PROGRAM PRG_HmiStatus
VAR
    fbBlinkTimer    : TON;
    bBlinkTimerQOld : BOOL;
    bFlash          : BOOL;
    fbEL6910Diagnostics : FB_EL6910Diagnostics;
    uiHeatStakeReasonNestId : UINT;
    bHeatStakeReasonRejectPending : BOOL;
END_VAR

// Same 500 ms toggle used by the validated Silicone Station banner.
fbBlinkTimer(IN := NOT fbBlinkTimer.Q, PT := T#500MS);

IF fbBlinkTimer.Q AND NOT bBlinkTimerQOld THEN
    GVL_HMI.bBlink_1Hz := NOT GVL_HMI.bBlink_1Hz;
END_IF

bBlinkTimerQOld := fbBlinkTimer.Q;
bFlash := GVL_HMI.bBlink_1Hz;

GVL_HMI.stStatus.eMachineState := GVL_MASTER.stStatus.eMachineState;
GVL_HMI.stStatus.eIndexState := GVL_MASTER.stStatus.eIndexState;
GVL_HMI.stStatus.eIndexPosition := GVL_MASTER.stInputs.eIndexPosition;
GVL_HMI.stStatus.bReady := GVL_MASTER.stStatus.bReady;
GVL_HMI.stStatus.bBusy := GVL_MASTER.stStatus.bBusy;
GVL_HMI.stStatus.bFaulted := GVL_MASTER.stStatus.bFaulted;
GVL_HMI.stStatus.bTwoHandsSafe := GVL_MASTER.stInputs.bTwoHandsSafe;
// Physical operator-nest part-present indication.
// This is intentionally NOT derived from nest tracking/result state.
// It follows the real sensor immediately whenever the operator places/removes
// a part in the nest currently located at the operator position.
GVL_HMI.stStatus.bLoadingStationEaglePresent :=GVL_IO.stInputs.bLoadingStationEaglePresent;
GVL_HMI.stStatus.bLoadingStationPbupPresent := GVL_IO.stInputs.bLoadingStationPbupPresent;
GVL_HMI.stStatus.bRejectChutePartPresent := GVL_MASTER.stInputs.bRejectChutePartPresent;
GVL_HMI.stStatus.bHeatStakeEaglePresent := GVL_MASTER.stInputs.bHeatStakeEaglePresent;
GVL_HMI.stStatus.bHeatStakePatchPresent := GVL_MASTER.stInputs.bHeatStakePatchPresent;
GVL_HMI.stStatus.bPbupMagnetPresent := GVL_MASTER.stInputs.bPbupMagnetPresent;
GVL_HMI.stStatus.bIndexReady := GVL_MASTER.stInputs.bIndexReady;
GVL_HMI.stStatus.bIndexLocked := GVL_MASTER.stInputs.bIndexLocked;
GVL_HMI.stStatus.bIndexCompletedSensor := GVL_MASTER.stInputs.bIndexCompletedSensor;
GVL_HMI.stStatus.bMainDoorClosed := GVL_MASTER.stInputs.bMainDoorClosed;
GVL_HMI.stStatus.bMainDoorLocked := GVL_MASTER.stInputs.bMainDoorLocked;
GVL_HMI.stStatus.bStartButtonActive := GVL_MASTER.stInputs.bStartButton;
GVL_HMI.stStatus.bStopButtonActive := GVL_MASTER.stInputs.bStopButton;
GVL_HMI.stStatus.bResetButtonActive := GVL_MASTER.stInputs.bResetButton;
GVL_HMI.stStatus.bStartButtonLamp := GVL_MASTER.stOutputs.bLedStart;
GVL_HMI.stStatus.bUp24VPowerSupplyOk := GVL_MASTER.stInputs.bUp24VPowerSupplyOk;
GVL_HMI.stStatus.bUs24VPowerSupplyOk := GVL_MASTER.stInputs.bUs24VPowerSupplyOk;
GVL_HMI.stStatus.b48VPowerSupplyOk := GVL_MASTER.stInputs.b48VPowerSupplyOk;
GVL_HMI.stStatus.bMainDoorDiagnosticOk := GVL_MASTER.stInputs.bMainDoorDiagnosticOk;
GVL_HMI.stStatus.bMs6FeedbackOk := GVL_MASTER.stInputs.bMs6FeedbackOk;
GVL_HMI.stStatus.bAirExhausted := GVL_MASTER.stInputs.bAirExhausted;
GVL_HMI.stStatus.bLeftFlapSafe := GVL_MASTER.stInputs.stSafety.bLeftFlapSafe;
GVL_HMI.stStatus.bRightFlapSafe := GVL_MASTER.stInputs.stSafety.bRightFlapSafe;
GVL_HMI.stStatus.bEnableSettings := GVL_MASTER.stStatus.bEnableSetting;
GVL_HMI.stStatus.bAllStationsCommissioned := GVL_MASTER.stStatus.bAllStationsCommissioned;
GVL_HMI.stStatus.bAutoCycleAllowed := GVL_MASTER.stStatus.bAutoCycleAllowed;
GVL_HMI.stStatus.bPatchSupportRetracted := FALSE; // Retired status; no sensor is fitted.
GVL_HMI.stStatus.bPatchSupportExtended := FALSE; // Retired status; no sensor is fitted.


GVL_HMI.stStatus.bNest1Blocked := NOT GVL_Persistent.aNestEnabled[1];
GVL_HMI.stStatus.bNest2Blocked := NOT GVL_Persistent.aNestEnabled[2];
GVL_HMI.stStatus.bNest3Blocked := NOT GVL_Persistent.aNestEnabled[3];
GVL_HMI.stStatus.bNest4Blocked := NOT GVL_Persistent.aNestEnabled[4];

GVL_HMI.stStatus.bDisabledNestPartIndexBlocked := GVL_MASTER.stStatus.bDisabledNestPartIndexBlocked;
GVL_HMI.stStatus.bDisabledNestPartPopupRequest :=GVL_MASTER.stStatus.bDisabledNestPartPopupRequest;
GVL_HMI.stStatus.uiDisabledNestPartPopupNestId :=GVL_MASTER.stStatus.uiDisabledNestPartPopupNestId;

GVL_HMI.stStatus.bRejectChuteFullLatched :=GVL_MASTER.stStatus.bRejectChuteFullLatched;
GVL_HMI.stStatus.bRejectChutePopupRequest :=GVL_MASTER.stStatus.bRejectChutePopupRequest;
GVL_HMI.stStatus.bRejectChuteStopRequest :=GVL_MASTER.stStatus.bRejectChuteStopRequest;
GVL_HMI.stStatus.bRejectChuteResetBlocked :=GVL_MASTER.stStatus.bRejectChuteResetBlocked;

GVL_HMI.stStatus.sRejectChutePopupMessage :=
    'Reject chute is full. Empty the reject chute and press Acknowledge.';

GVL_HMI.stStatus.bHeatStakeHeadUp := GVL_MASTER.stStatus.bHeatStakeHeadUp;
GVL_HMI.stStatus.bHeatStakeHeadDown := GVL_MASTER.stStatus.bHeatStakeHeadDown;
GVL_HMI.stStatus.bHeatStakeHeadDownTimeoutFault := GVL_MASTER.stStatus.bHeatStakeHeadDownTimeoutFault;
GVL_HMI.stStatus.bHeatStakeHeadUpTimeoutFault := GVL_MASTER.stStatus.bHeatStakeHeadUpTimeoutFault;
GVL_HMI.stStatus.bHeatStakeHeadSensorConflictFault := GVL_MASTER.stStatus.bHeatStakeHeadSensorConflictFault;

// Use the same TC3/head criterion as the machine's hot-door lock demand.
GVL_HMI.bUnlockDoorVisible :=
    (GVL_MASTER.stStatus.eMachineState = E_MachineState.Stopped)
    AND GVL_MASTER.stStatus.stMainDoorLock.bLockRequest
    AND NOT (GVL_MASTER.stStatus.stHeatStakeTemperature.rOverTempTemperatureC <
        GVL_Config.rMainDoorHotTemperatureLimitC);
// A stale hot-door popup must not remain open once the head cools or the state changes.
IF NOT GVL_HMI.bUnlockDoorVisible THEN
    GVL_HMI.bUnlockDoorPopupRequest := FALSE;
END_IF


IF (GVL_MASTER.stStatus.uiDisabledNestPartPopupNestId >= 1)
    AND (GVL_MASTER.stStatus.uiDisabledNestPartPopupNestId <= 4)
THEN
    GVL_HMI.stStatus.sDisabledNestPartPopupMessage :=
        CONCAT(
            CONCAT(
                'Nest ',
                UINT_TO_STRING(GVL_MASTER.stStatus.uiDisabledNestPartPopupNestId)
            ),
            ' is disabled. Remove the part from this nest before indexing.'
        );
ELSE
    GVL_HMI.stStatus.sDisabledNestPartPopupMessage :=
        'A disabled nest contains a part. Remove the part before indexing.';
END_IF

GVL_HMI.stStatus.stPatchDispense := GVL_MASTER.stStatus.stPatchDispense;
// Display aggregate Patch faults, including feeding/motion, without changing control state.
GVL_HMI.stStatus.stPatchDispense.bFault :=
    GVL_MASTER.stStatus.stPatchDispense.bFault
    OR GVL_Motion.stPatchFeedStatus.bFault
    OR GVL_Motion.AxisDriveMotor.bError;
IF GVL_MASTER.stStatus.eMachineState = E_MachineState.Manual THEN
    // Continuous UP holding at HOME is idle; actual manual actions are busy.
    GVL_HMI.stStatus.stPatchDispense.bBusy :=
        GVL_MASTER.stStatus.stPatchDispense.bBusy
        OR NOT GVL_MASTER.stStatus.stPatchDispense.bHome
        OR GVL_Motion.stPatchFeedStatus.bBusy
        OR GVL_Motion.AxisDriveMotor.bMoving
        OR GVL_MASTER.stOutputs.bPatchVerticalDown
        OR GVL_MASTER.stOutputs.bPatchDispenserAir;
    GVL_HMI.stStatus.stPatchDispense.bReady :=
        GVL_MASTER.stStatus.stPatchDispense.bCommissioned
        AND GVL_MASTER.stStatus.stPatchDispense.bHome
        AND NOT GVL_HMI.stStatus.stPatchDispense.bBusy
        AND NOT GVL_HMI.stStatus.stPatchDispense.bFault;
END_IF
// ReadyToStart indication accepts the deliberately disabled, idle M1 axis.
// This does not change FB readiness, motion enable or sequence start permissives.
IF GVL_MASTER.stStatus.eMachineState = E_MachineState.ReadyToStart THEN
    GVL_HMI.stStatus.stPatchDispense.bReady :=
        GVL_MASTER.stStatus.stPatchDispense.bCommissioned
        AND (GVL_MASTER.stStatus.stPatchDispense.eState = E_PatchStationState.Ready)
        AND GVL_MASTER.stStatus.stPatchDispense.bHome
        AND NOT GVL_MASTER.stStatus.stPatchDispense.bBusy
        AND NOT GVL_HMI.stStatus.stPatchDispense.bFault
        AND GVL_MASTER.stInputs.stSafety.bSafetyOk
        AND GVL_MASTER.stInputs.stSafety.bMotionSafetyPermitted
        AND GVL_MASTER.stInputs.bMainDoorClosed
        AND GVL_Safety.bAirSupplySafe
        AND NOT GVL_Motion.stPatchFeedStatus.bBusy
        AND NOT GVL_Motion.AxisDriveMotor.bMoving
        AND NOT GVL_Motion.AxisDriveMotor.Axis.Status.ErrorStop
        AND (GVL_Motion.AxisDriveMotor.Axis.NcToPlc.AxisId <> 0)
        AND (GVL_Motion.AxisDriveMotor.bStandstill
            OR GVL_Motion.AxisDriveMotor.Axis.Status.Disabled);
END_IF
GVL_HMI.stStatus.stHeatStake := GVL_MASTER.stStatus.stHeatStake;
GVL_HMI.stStatus.stHeatStakeTemperature := GVL_MASTER.stStatus.stHeatStakeTemperature;
GVL_HMI.stStatus.stHeatStakeProcess := GVL_MASTER.stStatus.stHeatStakeProcess;
GVL_HMI.stStatus.stHeatStakeProcessSettings := GVL_Persistent.stHeatStakeProcessSettings;
GVL_HMI.stStatus.bHeatStakeProcessSettingsWriteBusy := PRG_HeatStakeProcessSettings.bWriteBusy;
GVL_HMI.stStatus.bHeatStakeProcessSettingsWriteError := PRG_HeatStakeProcessSettings.bWriteError;
GVL_HMI.stStatus.udiHeatStakeProcessSettingsWriteErrorId := PRG_HeatStakeProcessSettings.udiWriteErrorId;
GVL_HMI.stStatus.stHeatStakeTemperatureSettings := GVL_Persistent.stHeatStakeTemperatureSettings;
GVL_HMI.stStatus.bHeatStakeSettingsApplyAccepted := PRG_HeatStakeTemperatureSettings.bApplyAccepted;
GVL_HMI.stStatus.bHeatStakeSettingsApplyRejected := PRG_HeatStakeTemperatureSettings.bApplyRejected;
GVL_HMI.stStatus.bHeatStakeSettingsWriteBusy := PRG_HeatStakeTemperatureSettings.bWriteBusy;
GVL_HMI.stStatus.bHeatStakeSettingsWriteError := PRG_HeatStakeTemperatureSettings.bWriteError;
GVL_HMI.stStatus.bHeatStakeSettingsSaveSuccessful := PRG_HeatStakeTemperatureSettings.bSaveSuccessful;
GVL_HMI.stStatus.bHeatStakeSettingsSaveFailed := PRG_HeatStakeTemperatureSettings.bSaveFailed;
GVL_HMI.stStatus.sHeatStakeSettingsApplyRejectReason := PRG_HeatStakeTemperatureSettings.sApplyRejectReason;
GVL_HMI.stStatus.udiHeatStakeSettingsWriteErrorId := PRG_HeatStakeTemperatureSettings.udiWriteErrorId;

// Manual-mode indexer station/nest display.
GVL_HMI.stStatus.uiPatchDispenseNestId := GVL_MASTER.stStatus.uiPatchDispenseNestId;
GVL_HMI.stStatus.uiHeatStakeNestId := GVL_MASTER.stStatus.uiHeatStakeNestId;
GVL_HMI.stStatus.uiVisionNestId := GVL_MASTER.stStatus.uiVisionNestId;

GVL_HMI.stStatus.bHeatStakeManualEnableAllowed := GVL_MASTER.stStatus.bHeatStakeManualEnableAllowed;
GVL_HMI.stStatus.bHeatStakeManualStakeAllowed := GVL_MASTER.stStatus.bHeatStakeManualStakeAllowed;
GVL_HMI.stStatus.bHeatStakeManualUnlockAllowed := GVL_MASTER.stStatus.bHeatStakeManualUnlockAllowed;
GVL_HMI.stStatus.bHeatStakeManualLockAllowed := GVL_MASTER.stStatus.bHeatStakeManualLockAllowed;
GVL_HMI.stStatus.bHeatStakeManualHeadDownAllowed := GVL_MASTER.stStatus.bHeatStakeManualHeadDownAllowed;
GVL_HMI.stStatus.bHeatStakeManualHeadUpAllowed := GVL_MASTER.stStatus.bHeatStakeManualHeadUpAllowed;
GVL_HMI.stStatus.bHeatStakeManualSupportAllowed := GVL_MASTER.stStatus.bHeatStakeManualSupportAllowed;
GVL_HMI.stStatus.bHeatStakeManualActionBusy := GVL_MASTER.stStatus.bHeatStakeManualActionBusy;
GVL_HMI.stStatus.bHeatStakeManualHeadUnlocked := GVL_MASTER.stStatus.bHeatStakeManualHeadUnlocked;

// Explain the published Stake Patch permission without changing control logic.
// Resolve the physical nest safely; do not index the array with an unknown ID.
uiHeatStakeReasonNestId := GVL_MASTER.stStatus.uiHeatStakeNestId;
bHeatStakeReasonRejectPending := FALSE;
IF (uiHeatStakeReasonNestId >= 1) AND (uiHeatStakeReasonNestId <= 4) THEN
    bHeatStakeReasonRejectPending :=
        GVL_MASTER.stStatus.aNest[uiHeatStakeReasonNestId].stHeatStakeResult.bValid
        AND (GVL_MASTER.stStatus.aNest[uiHeatStakeReasonNestId].stHeatStakeResult.udiAlertCode
            = GVL_MASTER.udiHeatStakePatchMissingAlertCode);
END_IF

// The permission is authoritative. Show one actionable blocking reason at a
// time; clearing it reveals the next remaining blocker. Never request a reset,
// acknowledge a reject or generate a movement from this presentation program.
IF GVL_MASTER.stStatus.bHeatStakeManualStakeAllowed THEN
    GVL_HMI.sHeatStakeManualStakeMessage := 'Ready - press Stake Patch';
ELSIF GVL_MASTER.stStatus.eMachineState <> E_MachineState.Manual THEN
    GVL_HMI.sHeatStakeManualStakeMessage := 'Machine not in Manual mode';
ELSIF NOT GVL_MASTER.stInputs.stSafety.bSafetyOk THEN
    GVL_HMI.sHeatStakeManualStakeMessage := 'Safety not ready';
ELSIF NOT GVL_MASTER.stCommand.bHeatStakeManualEnable THEN
    GVL_HMI.sHeatStakeManualStakeMessage := 'Enable Heat Stake';
ELSIF GVL_MASTER.stStatus.bRejectChuteStopRequest THEN
    GVL_HMI.sHeatStakeManualStakeMessage := 'Reject chute stop active';
ELSIF NOT GVL_MASTER.stStatus.stHeatStakeTemperature.bIndexTemperatureReady THEN
    IF GVL_MASTER.stStatus.stHeatStakeTemperature.bFault THEN
        GVL_HMI.sHeatStakeManualStakeMessage := 'Temperature fault - see alarms';
    ELSE
        GVL_HMI.sHeatStakeManualStakeMessage := 'Temperature not ready';
    END_IF
ELSIF GVL_MASTER.stStatus.stHeatStake.bFault THEN
    GVL_HMI.sHeatStakeManualStakeMessage := 'Heat Stake fault - see alarms';
ELSIF NOT GVL_MASTER.stStatus.stHeatStake.bCommissioned THEN
    GVL_HMI.sHeatStakeManualStakeMessage := 'Heat Stake disabled - engineering check';
ELSIF GVL_MASTER.stStatus.bHeatStakeManualActionBusy THEN
    GVL_HMI.sHeatStakeManualStakeMessage := 'Manual head action running';
ELSIF GVL_MASTER.stStatus.stHeatStake.eState = E_PatchStationState.Processing THEN
    GVL_HMI.sHeatStakeManualStakeMessage := 'Heat Stake cycle running';
ELSIF NOT GVL_MASTER.stInputs.bStation2SupportRetracted THEN
    GVL_HMI.sHeatStakeManualStakeMessage := 'Retract nest support';
ELSIF NOT GVL_MASTER.stInputs.bHeatStakeHeadUp OR GVL_MASTER.stInputs.bHeatStakeHeadDown THEN
    GVL_HMI.sHeatStakeManualStakeMessage := 'Head not confirmed UP';
ELSIF GVL_MASTER.stStatus.bHeatStakeManualHeadUnlocked THEN
    GVL_HMI.sHeatStakeManualStakeMessage := 'Head marked UNLOCKED - use Lock';
ELSIF bHeatStakeReasonRejectPending THEN
    GVL_HMI.sHeatStakeManualStakeMessage := CONCAT(
        CONCAT('Nest ', UINT_TO_STRING(uiHeatStakeReasonNestId)), ': reject confirmation pending');
ELSIF NOT GVL_MASTER.stInputs.bHeatStakeEaglePresent THEN
    GVL_HMI.sHeatStakeManualStakeMessage := 'Part not detected at Heat Stake';
ELSIF GVL_MASTER.stStatus.stIndexStatus.bBusy THEN
    GVL_HMI.sHeatStakeManualStakeMessage := 'Index table busy';
ELSIF GVL_MASTER.stStatus.stHeatStake.eState = E_PatchStationState.Complete THEN
    GVL_HMI.sHeatStakeManualStakeMessage := 'Cycle complete - awaiting reset';
ELSIF GVL_MASTER.stStatus.stHeatStake.bBusy THEN
    GVL_HMI.sHeatStakeManualStakeMessage := 'Heat Stake busy - see diagnostics';
ELSIF NOT GVL_MASTER.stStatus.stHeatStake.bReady THEN
    GVL_HMI.sHeatStakeManualStakeMessage := 'Heat Stake not ready - see diagnostics';
ELSE
    // Publication and permission may straddle a one-scan state transition.
    GVL_HMI.sHeatStakeManualStakeMessage := 'Permissive updating - wait';
END_IF


// =====================================================
// VISION MANUAL MODE
// =====================================================

// General manual enable permissive
GVL_HMI.stStatus.bVisionManualEnableAllowed :=GVL_MASTER.stStatus.bVisionManualEnableAllowed;
GVL_HMI.stStatus.bVisionManualRunSequenceAllowed :=GVL_MASTER.stStatus.bVisionManualRunSequenceAllowed;
// Vision Manual Mode - Home
GVL_HMI.stStatus.bVisionManualHomeAllowed :=GVL_MASTER.stStatus.bVisionManualHomeAllowed;
GVL_HMI.stStatus.bVisionHome :=GVL_MASTER.stStatus.bVisionHome;

// -----------------------------------------------------
// Horizontal
// -----------------------------------------------------

GVL_HMI.stStatus.bVisionHorizontalBackAllowed :=
    GVL_MASTER.stStatus.bVisionHorizontalBackAllowed;

GVL_HMI.stStatus.bVisionHorizontalFrontAllowed :=
    GVL_MASTER.stStatus.bVisionHorizontalFrontAllowed;

GVL_HMI.stStatus.bVisionHorizontalBack :=
    GVL_MASTER.stStatus.bVisionHorizontalBack;

GVL_HMI.stStatus.bVisionHorizontalFront :=
    GVL_MASTER.stStatus.bVisionHorizontalFront;


// -----------------------------------------------------
// Vertical
// -----------------------------------------------------

GVL_HMI.stStatus.bVisionVerticalUpAllowed :=
    GVL_MASTER.stStatus.bVisionVerticalUpAllowed;

GVL_HMI.stStatus.bVisionVerticalIntermediateAllowed := FALSE; // Retired compatibility field.

GVL_HMI.stStatus.bVisionVerticalFullDownAllowed :=
    GVL_MASTER.stStatus.bVisionVerticalFullDownAllowed;

GVL_HMI.stStatus.bVisionVerticalUp :=
    GVL_MASTER.stStatus.bVisionVerticalUp;

GVL_HMI.stStatus.bVisionVerticalDown :=
    GVL_MASTER.stStatus.bVisionVerticalDown;


// -----------------------------------------------------
// Gripper
// -----------------------------------------------------

GVL_HMI.stStatus.bVisionGripOpenAllowed :=
    GVL_MASTER.stStatus.bVisionGripOpenAllowed;

GVL_HMI.stStatus.bVisionGripCloseAllowed :=
    GVL_MASTER.stStatus.bVisionGripCloseAllowed;

GVL_HMI.stStatus.bVisionGripOpen :=
    GVL_MASTER.stStatus.bVisionGripOpen;

GVL_HMI.stStatus.bVisionGripClosed :=
    GVL_MASTER.stStatus.bVisionGripClosed;


// -----------------------------------------------------
// Rotation
// -----------------------------------------------------

GVL_HMI.stStatus.bVisionRotate0Allowed :=GVL_MASTER.stStatus.bVisionRotate0Allowed;
GVL_HMI.stStatus.bVisionRotate180Allowed := GVL_MASTER.stStatus.bVisionRotate180Allowed;
GVL_HMI.stStatus.bVisionRotate0 :=GVL_MASTER.stStatus.bVisionRotate0;
GVL_HMI.stStatus.bVisionRotate180 :=GVL_MASTER.stStatus.bVisionRotate180;


// -----------------------------------------------------
// Support
// -----------------------------------------------------

GVL_HMI.stStatus.bVisionSupportAllowed := FALSE; // Retired compatibility field.
GVL_HMI.stStatus.bVisionSupportExtended := FALSE; // Retired compatibility field.
GVL_HMI.stStatus.bVisionSupportRetracted := FALSE; // Retired compatibility field.


// -----------------------------------------------------
// Vision station status
// -----------------------------------------------------

GVL_HMI.stStatus.stVision :=GVL_MASTER.stStatus.stVision;
GVL_HMI.stStatus.eOperatorInstruction := GVL_MASTER.stStatus.eOperatorInstruction;
GVL_HMI.stStatus.stOperatorStation := GVL_MASTER.stStatus.stOperatorStation;
GVL_HMI.stStatus.aNest := GVL_MASTER.stStatus.aNest;

// Dedicated operator message remains available for a dedicated HMI label.
GVL_HMI.stStatus.sOperatorMessage := GVL_MASTER.stStatus.sOperatorMessage;

// Keep compatibility with the existing message control inherited from
// Silicone: during AutoCycle, show the operator instruction in the main
// message field when one is active.


// =====================================================
// TEST HISTORY
// =====================================================
// Publish the persistent Test History to the HMI.
// Production Statistics reset does not affect this data.

GVL_HMI.astTestHistory := GVL_Persistent.astTestHistory;

GVL_HMI.uiTestHistoryWriteIndex :=
    GVL_Persistent.uiTestHistoryWriteIndex;

GVL_HMI.uiTestHistoryCount :=
    GVL_Persistent.uiTestHistoryCount;
	

IF GVL_MASTER.stStatus.eMachineState = E_MachineState.Dwell THEN

    // Show live heater temperature in the main HMI message.
    GVL_HMI.stStatus.sMachineMessage :=
        GVL_MASTER.stStationEvents[3].aEvents[12].bEventText;

ELSIF (GVL_MASTER.stStatus.eMachineState = E_MachineState.AutoCycle)
    AND (LEN(GVL_MASTER.stStatus.sOperatorMessage) > 0)
THEN

    GVL_HMI.stStatus.sMachineMessage :=
        GVL_MASTER.stStatus.sOperatorMessage;

ELSE

    GVL_HMI.stStatus.sMachineMessage :=
        GVL_MASTER.stStatus.sMachineMessage;

END_IF

GVL_HMI.stStatus.sAutoCycleBlockReason := GVL_MASTER.stStatus.sAutoCycleBlockReason;
GVL_HMI.stStatistics.aNest := GVL_MASTER.stStatus.aNestStatistics;
CASE GVL_MASTER.stInputs.eIndexPosition OF
    E_TablePosition.Position1: GVL_HMI.stStatus.iNestRotationAngle := 0;
    E_TablePosition.Position2: GVL_HMI.stStatus.iNestRotationAngle := 270;
    E_TablePosition.Position3: GVL_HMI.stStatus.iNestRotationAngle := 180;
    E_TablePosition.Position4: GVL_HMI.stStatus.iNestRotationAngle := 90;
ELSE GVL_HMI.stStatus.iNestRotationAngle := 0;
END_CASE




CASE GVL_MASTER.stStatus.eMachineState OF
    E_MachineState.PowerUp: GVL_HMI.StatusHMI.sMachineStatusText := 'SYSTEM POWER UP'; GVL_HMI.StatusHMI.sBannerBckColor := GVL_HMI.sYELLOW; GVL_HMI.StatusHMI.sBannerTextColor := GVL_HMI.sBLACK;
    E_MachineState.Initialising: GVL_HMI.StatusHMI.sMachineStatusText := 'SYSTEM INITIALIZING'; GVL_HMI.StatusHMI.sBannerBckColor := GVL_HMI.sYELLOW; GVL_HMI.StatusHMI.sBannerTextColor := GVL_HMI.sBLACK;
    E_MachineState.ReadyToStart:
        GVL_HMI.StatusHMI.sMachineStatusText := 'SYSTEM READY TO START';
        IF bFlash THEN
            GVL_HMI.StatusHMI.sBannerBckColor := GVL_HMI.sGREEN;
            GVL_HMI.StatusHMI.sBannerTextColor := GVL_HMI.sWHITE;
        ELSE
            GVL_HMI.StatusHMI.sBannerBckColor := GVL_HMI.sWHITE;
            GVL_HMI.StatusHMI.sBannerTextColor := GVL_HMI.sGREEN;
        END_IF
	
	E_MachineState.Dwell:
		GVL_HMI.StatusHMI.sMachineStatusText :='DWELL'; GVL_HMI.StatusHMI.sBannerBckColor := GVL_HMI.sORANGE; GVL_HMI.StatusHMI.sBannerTextColor := GVL_HMI.sWHITE;
    E_MachineState.AutoCycle: 
			GVL_HMI.StatusHMI.sMachineStatusText := 'SYSTEM AUTO CYCLE'; GVL_HMI.StatusHMI.sBannerBckColor := GVL_HMI.sGREEN; GVL_HMI.StatusHMI.sBannerTextColor := GVL_HMI.sWHITE;
	E_MachineState.Stopping: 
			GVL_HMI.StatusHMI.sMachineStatusText := 'STOPPING'; GVL_HMI.StatusHMI.sBannerBckColor := GVL_HMI.sGREY; GVL_HMI.StatusHMI.sBannerTextColor := GVL_HMI.sWHITE;
    E_MachineState.Stopped: 
			GVL_HMI.StatusHMI.sMachineStatusText := 'CYCLE STOPPED'; GVL_HMI.StatusHMI.sBannerBckColor := GVL_HMI.sGREY; GVL_HMI.StatusHMI.sBannerTextColor := GVL_HMI.sWHITE;
    E_MachineState.Fault:
        	GVL_HMI.StatusHMI.sMachineStatusText := 'IMMEDIATE FAULT';
			
			
        IF bFlash THEN
            GVL_HMI.StatusHMI.sBannerBckColor := GVL_HMI.sREDFail;
            GVL_HMI.StatusHMI.sBannerTextColor := GVL_HMI.sWHITE;
        ELSE
            GVL_HMI.StatusHMI.sBannerBckColor := GVL_HMI.sWHITE;
            GVL_HMI.StatusHMI.sBannerTextColor := GVL_HMI.sREDFail;
        END_IF
    E_MachineState.Manual: GVL_HMI.StatusHMI.sMachineStatusText := 'MANUAL MODE'; GVL_HMI.StatusHMI.sBannerBckColor := GVL_HMI.sBLUEInProgress; GVL_HMI.StatusHMI.sBannerTextColor := GVL_HMI.sWHITE;
END_CASE
// Native terminal diagnostics: retain each terminal own ST_Terminal_Info instance.
GVL_EtherCAT.stTerm1_EK1100.stTerminalInfo.fbTerminalInfo(
    nTerminalState := GVL_EtherCAT.stTerm1_EK1100.stTerminalInfo.nTerminal_State,
    sTerminalState => GVL_EtherCAT.stTerm1_EK1100.stTerminalInfo.sTerminalInfo,
    bTerminalOperational => GVL_EtherCAT.stTerm1_EK1100.stTerminalInfo.bTerminalOperational);
GVL_EtherCAT.stTerm2_EL6070.stTerminalInfo.fbTerminalInfo(
    nTerminalState := GVL_EtherCAT.stTerm2_EL6070.stTerminalInfo.nTerminal_State,
    sTerminalState => GVL_EtherCAT.stTerm2_EL6070.stTerminalInfo.sTerminalInfo,
    bTerminalOperational => GVL_EtherCAT.stTerm2_EL6070.stTerminalInfo.bTerminalOperational);
GVL_EtherCAT.stTerm3_EL6910.stTerminalInfo.fbTerminalInfo(
    nTerminalState := GVL_EtherCAT.stTerm3_EL6910.stTerminalInfo.nTerminal_State,
    sTerminalState => GVL_EtherCAT.stTerm3_EL6910.stTerminalInfo.sTerminalInfo,
    bTerminalOperational => GVL_EtherCAT.stTerm3_EL6910.stTerminalInfo.bTerminalOperational);
GVL_EtherCAT.stTerm4_EL1918.stTerminalInfo.fbTerminalInfo(
    nTerminalState := GVL_EtherCAT.stTerm4_EL1918.stTerminalInfo.nTerminal_State,
    sTerminalState => GVL_EtherCAT.stTerm4_EL1918.stTerminalInfo.sTerminalInfo,
    bTerminalOperational => GVL_EtherCAT.stTerm4_EL1918.stTerminalInfo.bTerminalOperational);
GVL_EtherCAT.stTerm5_EL1918.stTerminalInfo.fbTerminalInfo(
    nTerminalState := GVL_EtherCAT.stTerm5_EL1918.stTerminalInfo.nTerminal_State,
    sTerminalState => GVL_EtherCAT.stTerm5_EL1918.stTerminalInfo.sTerminalInfo,
    bTerminalOperational => GVL_EtherCAT.stTerm5_EL1918.stTerminalInfo.bTerminalOperational);
GVL_EtherCAT.stTerm6_EL2904.stTerminalInfo.fbTerminalInfo(
    nTerminalState := GVL_EtherCAT.stTerm6_EL2904.stTerminalInfo.nTerminal_State,
    sTerminalState => GVL_EtherCAT.stTerm6_EL2904.stTerminalInfo.sTerminalInfo,
    bTerminalOperational => GVL_EtherCAT.stTerm6_EL2904.stTerminalInfo.bTerminalOperational);
GVL_EtherCAT.stTerm7_EL1809.stTerminalInfo.fbTerminalInfo(
    nTerminalState := GVL_EtherCAT.stTerm7_EL1809.stTerminalInfo.nTerminal_State,
    sTerminalState => GVL_EtherCAT.stTerm7_EL1809.stTerminalInfo.sTerminalInfo,
    bTerminalOperational => GVL_EtherCAT.stTerm7_EL1809.stTerminalInfo.bTerminalOperational);
GVL_EtherCAT.stTerm8_EL1809.stTerminalInfo.fbTerminalInfo(
    nTerminalState := GVL_EtherCAT.stTerm8_EL1809.stTerminalInfo.nTerminal_State,
    sTerminalState => GVL_EtherCAT.stTerm8_EL1809.stTerminalInfo.sTerminalInfo,
    bTerminalOperational => GVL_EtherCAT.stTerm8_EL1809.stTerminalInfo.bTerminalOperational);
GVL_EtherCAT.stTerm9_EL2809.stTerminalInfo.fbTerminalInfo(
    nTerminalState := GVL_EtherCAT.stTerm9_EL2809.stTerminalInfo.nTerminal_State,
    sTerminalState => GVL_EtherCAT.stTerm9_EL2809.stTerminalInfo.sTerminalInfo,
    bTerminalOperational => GVL_EtherCAT.stTerm9_EL2809.stTerminalInfo.bTerminalOperational);
GVL_EtherCAT.stTerm10_EL2809.stTerminalInfo.fbTerminalInfo(
    nTerminalState := GVL_EtherCAT.stTerm10_EL2809.stTerminalInfo.nTerminal_State,
    sTerminalState => GVL_EtherCAT.stTerm10_EL2809.stTerminalInfo.sTerminalInfo,
    bTerminalOperational => GVL_EtherCAT.stTerm10_EL2809.stTerminalInfo.bTerminalOperational);
GVL_EtherCAT.stTerm11_EL3058.stTerminalInfo.fbTerminalInfo(
    nTerminalState := GVL_EtherCAT.stTerm11_EL3058.stTerminalInfo.nTerminal_State,
    sTerminalState => GVL_EtherCAT.stTerm11_EL3058.stTerminalInfo.sTerminalInfo,
    bTerminalOperational => GVL_EtherCAT.stTerm11_EL3058.stTerminalInfo.bTerminalOperational);
GVL_EtherCAT.stTerm12_EL9410.stTerminalInfo.fbTerminalInfo(
    nTerminalState := GVL_EtherCAT.stTerm12_EL9410.stTerminalInfo.nTerminal_State,
    sTerminalState => GVL_EtherCAT.stTerm12_EL9410.stTerminalInfo.sTerminalInfo,
    bTerminalOperational => GVL_EtherCAT.stTerm12_EL9410.stTerminalInfo.bTerminalOperational);
GVL_EtherCAT.stTerm13_EL2502.stTerminalInfo.fbTerminalInfo(
    nTerminalState := GVL_EtherCAT.stTerm13_EL2502.stTerminalInfo.nTerminal_State,
    sTerminalState => GVL_EtherCAT.stTerm13_EL2502.stTerminalInfo.sTerminalInfo,
    bTerminalOperational => GVL_EtherCAT.stTerm13_EL2502.stTerminalInfo.bTerminalOperational);
GVL_EtherCAT.stTerm14_EL9576.stTerminalInfo.fbTerminalInfo(
    nTerminalState := GVL_EtherCAT.stTerm14_EL9576.stTerminalInfo.nTerminal_State,
    sTerminalState => GVL_EtherCAT.stTerm14_EL9576.stTerminalInfo.sTerminalInfo,
    bTerminalOperational => GVL_EtherCAT.stTerm14_EL9576.stTerminalInfo.bTerminalOperational);
GVL_EtherCAT.stTerm15_EL7201.stTerminalInfo.fbTerminalInfo(
    nTerminalState := GVL_EtherCAT.stTerm15_EL7201.stTerminalInfo.nTerminal_State,
    sTerminalState => GVL_EtherCAT.stTerm15_EL7201.stTerminalInfo.sTerminalInfo,
    bTerminalOperational => GVL_EtherCAT.stTerm15_EL7201.stTerminalInfo.bTerminalOperational);
GVL_EtherCAT.stTerm16_EL7201.stTerminalInfo.fbTerminalInfo(
    nTerminalState := GVL_EtherCAT.stTerm16_EL7201.stTerminalInfo.nTerminal_State,
    sTerminalState => GVL_EtherCAT.stTerm16_EL7201.stTerminalInfo.sTerminalInfo,
    bTerminalOperational => GVL_EtherCAT.stTerm16_EL7201.stTerminalInfo.bTerminalOperational);
GVL_EtherCAT.stTerm17_EL7201.stTerminalInfo.fbTerminalInfo(
    nTerminalState := GVL_EtherCAT.stTerm17_EL7201.stTerminalInfo.nTerminal_State,
    sTerminalState => GVL_EtherCAT.stTerm17_EL7201.stTerminalInfo.sTerminalInfo,
    bTerminalOperational => GVL_EtherCAT.stTerm17_EL7201.stTerminalInfo.bTerminalOperational);
GVL_EtherCAT.stTerm18_EL2904.stTerminalInfo.fbTerminalInfo(
    nTerminalState := GVL_EtherCAT.stTerm18_EL2904.stTerminalInfo.nTerminal_State,
    sTerminalState => GVL_EtherCAT.stTerm18_EL2904.stTerminalInfo.sTerminalInfo,
    bTerminalOperational => GVL_EtherCAT.stTerm18_EL2904.stTerminalInfo.bTerminalOperational);
GVL_EtherCAT.stTerm19_EL1809.stTerminalInfo.fbTerminalInfo(
    nTerminalState := GVL_EtherCAT.stTerm19_EL1809.stTerminalInfo.nTerminal_State,
    sTerminalState => GVL_EtherCAT.stTerm19_EL1809.stTerminalInfo.sTerminalInfo,
    bTerminalOperational => GVL_EtherCAT.stTerm19_EL1809.stTerminalInfo.bTerminalOperational);
GVL_EtherCAT.stTerm20_EL4022.stTerminalInfo.fbTerminalInfo(
    nTerminalState := GVL_EtherCAT.stTerm20_EL4022.stTerminalInfo.nTerminal_State,
    sTerminalState => GVL_EtherCAT.stTerm20_EL4022.stTerminalInfo.sTerminalInfo,
    bTerminalOperational => GVL_EtherCAT.stTerm20_EL4022.stTerminalInfo.bTerminalOperational);
GVL_EtherCAT.stTerm21_EL3314.stTerminalInfo.fbTerminalInfo(
    nTerminalState := GVL_EtherCAT.stTerm21_EL3314.stTerminalInfo.nTerminal_State,
    sTerminalState => GVL_EtherCAT.stTerm21_EL3314.stTerminalInfo.sTerminalInfo,
    bTerminalOperational => GVL_EtherCAT.stTerm21_EL3314.stTerminalInfo.bTerminalOperational);
GVL_EtherCAT.stTerm22_EL6633.stTerminalInfo.fbTerminalInfo(
    nTerminalState := GVL_EtherCAT.stTerm22_EL6633.stTerminalInfo.nTerminal_State,
    sTerminalState => GVL_EtherCAT.stTerm22_EL6633.stTerminalInfo.sTerminalInfo,
    bTerminalOperational => GVL_EtherCAT.stTerm22_EL6633.stTerminalInfo.bTerminalOperational);
GVL_EtherCAT.stFestoTerminalInfo.fbTerminalInfo(
    nTerminalState := GVL_EtherCAT.stFestoTerminalInfo.nTerminal_State,
    sTerminalState => GVL_EtherCAT.stFestoTerminalInfo.sTerminalInfo,
    bTerminalOperational => GVL_EtherCAT.stFestoTerminalInfo.bTerminalOperational);

// EL6910 internal diagnostics only; no machine or TwinSAFE decisions consume these values.
fbEL6910Diagnostics(
    bEnable := GVL_EtherCAT.stTerm3_EL6910.stTerminalInfo.bTerminalOperational,
    sMasterNetId := '172.18.239.27.2.1',
    uiSlaveAddress := 1003,
    stStatus := GVL_EL6910Diagnostics.stStatus);

END_PROGRAM

(* stored: Version 1.1.0.1, ProductVersion 3.1.4026.18
   POU PRG_HmiStatus: Id {4da5e538-fb78-4127-b5c1-141c740c9ced}, SpecialFunc None *)
